PROGRAM MAIN
VAR
END_VAR

END_PROGRAM

(* stored: Version 1.1.0.1
   POU MAIN: Id {6ef588eb-c0b5-4164-a8cc-ee299a078164} *)
